FUNCTION_BLOCK Protection
VAR_IN_OUT
	axis  		: ARRAY [XP .. XM] OF AxisGroup;
	stateLVL1 	: INT;
	speed 		: LREAL;
END_VAR
VAR_INPUT
	reset : BOOL;
END_VAR
VAR_OUTPUT
END_VAR
VAR
	checkHomed_TON 	: TON;
	
	//for use end of travel protection
	eotDistTravel	: ARRAY [XP .. XM, lmHome .. lmDeploy] OF LREAL;
	eotDistStart	: ARRAY [XP .. XM, lmHome .. lmDeploy] OF LREAL;
	eotRtrig		: ARRAY [XP .. XM, lmHome .. lmDeploy] OF R_Trig;
END_VAR

VAR CONSTANT
	XP 			: INT 	:= 0;
	XM 			: INT 	:= 1;
	lmHome 		: INT 	:= 0;
	lmDeploy	: INT 	:= 1;
	eotTravelLm	: LREAL := 2;
	diffLimit 	: LREAL	:= 5;
END_VAR

(*
This function block contains the logic for the shutter system protection. 
*)


//Brake status check - if brakes are not disengaged, disable axis movement
IF axis[XP].brake AND axis[XM].brake THEN 
	axis[XP].mcPower(Axis := axis[XP].axisRef, Enable := TRUE, Enable_Positive := TRUE, Enable_Negative := TRUE);
	axis[XM].mcPower(Axis := axis[XM].axisRef, Enable := TRUE, Enable_Positive := TRUE, Enable_Negative := TRUE);	
ELSE
	axis[XP].mcPower(Axis := axis[XP].axisRef, Enable := TRUE, Enable_Positive := FALSE, Enable_Negative := FALSE);
	axis[XM].mcPower(Axis := axis[XM].axisRef, Enable := TRUE, Enable_Positive := FALSE, Enable_Negative := FALSE); 
END_IF

//Prevents movement if not homed.
(*
IF stateLVL1>400 THEN
	IF NOT axis[XP].axisRef.Status.Homed OR NOT axis[XM].axisRef.Status.Homed THEN
		 axis[XP].mcStop(Axis:=axis[XP].axisRef, Execute:=TRUE);
		 axis[XM].mcStop(Axis:=axis[XM].axisRef, Execute:=TRUE);
		//To-Do later... Add error code for not homed
	END_IF
END_IF
*)

//Check for calibration. If not both blades not calibrated, speed cannot be higher than 200 mms.
IF NOT axis[XP].isCalibrated AND NOT axis[XM].isCalibrated THEN
	IF speed > 200 THEN
		speed := 0;
	END_IF
END_IF

//Compare position seen by hall switch with position seen by motor encoder
IF axis[XP].isCalibrated AND axis[XM].isCalibrated THEN
	IF ABS(axis[XP].posDiffAtTrip)>diffLimit OR ABS(axis[XM].posDiffAtTrip)>diffLimit THEN
		axis[XP].mcStop(Axis := axis[XP].axisRef, Execute := TRUE);
		axis[XM].mcStop(Axis := axis[XM].axisRef, Execute := TRUE);
	END_IF
END_IF


(* limit switch protection no enabled; require all limit switch to function ....	
//End of travel stop
eotRtrig[XP,lmHome](CLK := axis[XM].limitHome);
eotRtrig[XP,lmDeploy](CLK := axis[XP].limitDeployed);
eotRtrig[XM,lmHome](CLK := axis[XM].limitHome);
eotRtrig[XM,lmDeploy](CLK := axis[XM].limitDeployed);
IF eotRtrig[XP,lmHome].Q THEN
	eotDistStart[XP,lmHome] := axis[XP].axisRef.NcToPlc.ActPos;
END_IF
IF eotRtrig[XP,lmDeploy].Q THEN
	eotDistStart[XP,lmDeploy] := axis[XP].axisRef.NcToPlc.ActPos;
END_IF
IF eotRtrig[XM,lmHome].Q THEN
	eotDistStart[XM,lmHome] := axis[XM].axisRef.NcToPlc.ActPos;
END_IF
IF eotRtrig[XM,lmDeploy].Q THEN
	eotDistStart[XM,lmDeploy] := axis[XM].axisRef.NcToPlc.ActPos;
END_IF

IF axis[XP].limitHome THEN
	eotDistTravel[XP,lmHome] := eotDistStart[XP,lmHome] - axis[XP].axisRef.NcToPlc.ActPos;
	IF eotDistTravel[XP,lmHome] > eotTravelLm THEN
		axis[XP].mcPower(Axis := axis[XP].axisRef, Enable_Negative := FALSE);
	END_IF
ELSE
	axis[XP].mcPower(Axis := axis[XP].axisRef, Enable_Negative := TRUE);
END_IF

IF axis[XP].limitDeployed THEN
	eotDistTravel[XP,lmDeploy] := axis[XP].axisRef.NcToPlc.ActPos - eotDistStart[XP,lmDeploy];
	IF eotDistTravel[XP,lmHome] > eotTravelLm THEN
		axis[XP].mcPower(Axis := axis[XP].axisRef, Enable_Positive := FALSE);
	END_IF
ELSE
	axis[XP].mcPower(Axis := axis[XP].axisRef, Enable_Positive := TRUE);
END_IF


IF axis[XM].limitHome THEN
	eotDistTravel[XM,lmHome] := axis[XM].axisRef.NcToPlc.ActPos - eotDistStart[XM,lmHome];
	IF eotDistTravel[XM,lmHome] > eotTravelLm THEN
		axis[XM].mcPower(Axis := axis[XM].axisRef, Enable_Positive := FALSE);
	END_IF
ELSE
	axis[XM].mcPower(Axis := axis[XM].axisRef, Enable_Positive := TRUE);
END_IF

IF axis[XM].limitDeployed THEN
	eotDistTravel[XM,lmDeploy] := eotDistStart[XM,lmDeploy] - axis[XM].axisRef.NcToPlc.ActPos;
	IF eotDistTravel[XM,lmHome] > eotTravelLm THEN
		axis[XM].mcPower(Axis := axis[XM].axisRef, Enable_Negative := FALSE);
	END_IF
ELSE
	axis[XM].mcPower(Axis := axis[XM].axisRef, Enable_Negative := TRUE);
END_IF

*)

END_FUNCTION_BLOCK

(* stored: Version 1.1.0.1, ProductVersion 3.1.4020.12
   POU Protection: Id {2dceb2c7-c1a1-4d57-b0b3-835d45fe31c4}, SpecialFunc None *)
